INTERFACE ITF_Group2 EXTENDS ITF_BaseGroupElement

END_INTERFACE

(* stored: Version 1.1.0.1
   Itf ITF_Group2: Id {41af1ba0-dc48-0a1a-181f-1bd4cd827794} *)
